// TIA Portal V20 export
TYPE "typeUnitCommunicationControlNodeBA040"
// stored: Namespace Unit1.Em2
   STRUCT
      noInterference { ExternalWritable := 'False'} : Bool;
      requestClamp { ExternalWritable := 'False'} : Bool;
      partOn { ExternalWritable := 'False'} : Bool;
      loadComplete { ExternalWritable := 'False'} : Bool;
   END_STRUCT;
END_TYPE
